(* IEC 61131-3 sources: codesys-build/examples/frame-assembly/src/io, 1 file *)

(* ---- PRG_ReadInputs.st ---- *)
PROGRAM PRG_ReadInputs
VAR
	Cycles : UDINT;
END_VAR
Cycles := Cycles + 1;
END_PROGRAM
